TYPE KeyAndValue :
STRUCT
	Key : STRING;
	Value : string;
END_STRUCT
END_TYPE

(* stored: Version 1.1.0.1, ProductVersion 3.1.4024.12
   DUT KeyAndValue: Id {dd492d75-630f-45ce-a83c-b4fabc88c7c1} *)
